// TIA Portal V19 export
ORGANIZATION_BLOCK "Main"   // OB1, FBD, ProgramCycle
TITLE = "Main Program Sweep (Cycle)"
   VAR_TEMP
      OB1_EV_CLASS : Byte;   // Bits 0-3 = 1 (Coming event), Bits 4-7 = 1 (Event class 1)
      OB1_SCAN_1 : Byte;   // 1 (Cold restart scan 1 of OB 1), 3 (Scan 2-n of OB 1)
      OB1_PRIORITY : Byte;   // Priority of OB Execution
      OB1_OB_NUMBR : Byte;   // 1 (Organization block 1, OB1)
      OB1_RESERVED_1 : Byte;   // Reserved for system
      OB1_RESERVED_2 : Byte;   // Reserved for system
      OB1_PREV_CYCLE : Int;   // Cycle time of previous OB1 scan (milliseconds)
      OB1_MIN_CYCLE : Int;   // Minimum cycle time of OB1 (milliseconds)
      OB1_MAX_CYCLE : Int;   // Maximum cycle time of OB1 (milliseconds)
      OB1_DATE_TIME : Date_And_Time;   // Date and time OB1 started
   END_VAR
   VAR_TEMP   // added for the SCL form of the ladder/FBD networks
      _w1 : Bool;
   END_VAR
BEGIN

REGION Network 1
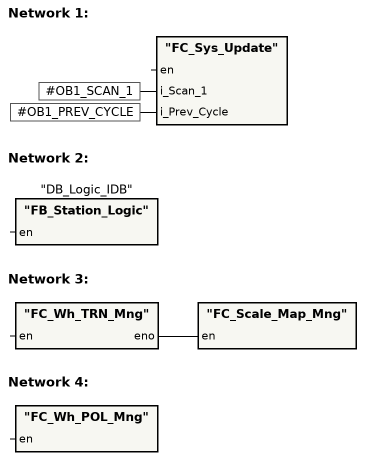
   "FC_Sys_Update"(i_Scan_1 := #OB1_SCAN_1, i_Prev_Cycle := #OB1_PREV_CYCLE);
END_REGION

REGION Network 2
   "DB_Logic_IDB"();   // "FB_Station_Logic"
END_REGION

REGION Network 3
   "FC_Wh_TRN_Mng"(ENO => #_w1);
   IF #_w1 THEN "FC_Scale_Map_Mng"(); END_IF;
END_REGION

REGION Network 4
   "FC_Wh_POL_Mng"();
END_REGION
END_ORGANIZATION_BLOCK
